PROGRAM MAIN
VAR
END_VAR

PLC_PRG();

END_PROGRAM

(* stored: Version 1.1.0.1, ProductVersion 3.1.4022.12
   POU MAIN: Id {a8fcc254-eba8-4599-a653-dce506a85a48}, SpecialFunc None *)
